Staubli VAL3: onF2Event.pgx

program onF2Event()
  local string l_sMessage
  local bool l_bYes
  local num i
begin
  // look if the bButton is enable
  if bButton[1]
    //
  endIf
end
